// TwinCAT 3 PLC project Nepionic_Log
// Title: Nepionic_Log
// Company: Nepionic
// Author: Nepionic
// ProjectVersion: 0.1.1
// ProgramVersion: 3.1.4026.22
// libraries:
//   Tc2_Standard, * (Beckhoff Automation GmbH)
//   Tc2_System, * (Beckhoff Automation GmbH)
//   Tc2_Utilities, * (Beckhoff Automation GmbH)
//   Tc3_DynamicMemory, * (Beckhoff Automation GmbH)
// project tree:
//   Lib/Appenders/AdsLog/ AdsLogAppender.TcPOU (not stored), LogLevelToAdsLogMsgType.TcPOU
//   Lib/Appenders/File/ DeleteFilesState.TcDUT (not stored), DeleteOldFiles.TcPOU, GenerateTimeData.TcPOU (not stored), GetFileAgeInSeconds.TcPOU (not stored), LoggingConfiguration.TcDUT, PersistToFileState.TcDUT (not stored), RollingIntervals.TcDUT (not stored)
//   Lib/Appenders/ LogAppender.TcIO (not stored)
//   Lib/ Constants.TcGVL, DateTime.TcPOU (not stored), Error.TcDUT (not stored), ErrorCodes.TcDUT (not stored)
//   Lib/Core/ LogAttribute.TcDUT, LogAttributeType.TcDUT (not stored), LogAttributeValueToString.TcPOU, LogLevel.TcDUT
//   Lib/Manager/ GetLogManager.TcPOU (not stored), LogManager.TcPOU (not stored)
//   Lib/Logger/ DefaultLogger.TcPOU, Logger.TcIO (not stored)
//   Lib/String/ AnyToString.TcPOU (not stored), DefaultStringBuilder.TcPOU (not stored), DynamicStringBuffer.TcPOU (not stored), LimitedStringBuilder.TcIO (not stored), StringBuilder.TcIO (not stored)

// ---- Lib/Appenders/File/LoggingConfiguration.TcDUT
// Configuration of TcLogCore
TYPE LoggingConfiguration :
STRUCT
	// File name where the logs should be written to. Should not include path.
	file_name : Tc2_System.T_MaxString;
	// File path where the logs should be written to. Will be prefixed to `FileName`
	file_path : Tc2_System.T_MaxString;
	// Whether to include the instance path of TcLog into the log message or not.
	include_instance_path : BOOL;
	/// Whether to write the logs to ADS output or not.
	write_to_ads : BOOL;
	/// Rolling interval: when to create a new log file.
	rolling_interval : RollingIntervals;
	/// What is the minimum log level that gets logged?
	minimum_level : LogLevel;
	/// Which delimiter should be used between the different parts of the log string?
	delimiter : STRING(1);
	/// When should old log files be deleted? Unit: days. Set it to `0` if log files should never be deleted. 
	log_file_life_span : UINT;
	/// Format of timestamp. See `TcLogCore.TimestampFormat` for formatting options.
	timestamp_format : STRING;
	/// Log only valid timestamps (skip log messages during time initialization (first few cycles)
	valid_timestamps_only: BOOL;
END_STRUCT
END_TYPE

// ---- Lib/Core/LogAttribute.TcDUT
// A single structured log attribute attached to a log entry.
//
// Binary layout (96 bytes, little-endian, matched by the Go otelcol-ads parser):
//   offset  0..31   key         STRING(31)            = 32 bytes  attribute name
//   offset 32       attr_type   LogAttributeType      =  1 byte   type tag
//   offset 33..95   value_bytes ARRAY[0..62] BYTE     = 63 bytes  payload (see attr_type)
//
// For attr_type = LogAttributeType.Str (11):
//   value_bytes holds a null-terminated STRING(62).
// For numeric/bool types, value_bytes[0..N-1] holds the value as little-endian bytes.
TYPE LogAttribute :
STRUCT
	// Attribute name, e.g. 'event.name', 'axis.speed'
	key : STRING(31);
	
	// Type tag — one of the LogAttrType enum values.
	attr_type : LogAttributeType;

	// Raw value bytes. Interpretation depends on attr_type.
	// For String: null-terminated string up to 62 chars.
	// For numeric/bool: little-endian encoded value in first N bytes.
	value_bytes : ARRAY[0..62] OF BYTE;
END_STRUCT
END_TYPE

// ---- Lib/Core/LogLevel.TcDUT
{attribute 'qualified_only'}
{attribute 'strict'}
{attribute 'to_string'}
TYPE LogLevel :
(
	Debug := 0,
	Information := 1,
	Warning := 2,
	Error := 3,
	Fatal := 4
);
END_TYPE

// ---- Lib/Constants.TcGVL
{attribute 'qualified_only'}
VAR_GLOBAL CONSTANT
	/// Fifo overhead needed to manage the string buffer
	FifoOverhead : UDINT := 10;
	/// Buffer size of temporary buffer used to persist all log messages in one cycle. 
	BufferSize : UDINT := (100 * (Tc2_System.MAX_STRING_LENGTH + FifoOverhead));
END_VAR

// ---- Lib/Appenders/AdsLog/LogLevelToAdsLogMsgType.TcPOU
// Converts TcLog.LogLevels into Tc2_System.AdsLog_MsgType_*.
{attribute 'hide'}
FUNCTION INTERNAL LogLevelToAdsLogMsgType : DWORD
VAR_INPUT
	log_level : LogLevel;
END_VAR
VAR
	return_value : DWORD;
END_VAR

CASE log_level OF
	LogLevel.Debug, LogLevel.Information:
		return_value := Tc2_System.AdsLog_MsgType_Hint;
		
	LogLevel.Warning:
		return_value := Tc2_System.AdsLog_MsgType_Warn;
		
	LogLevel.Error, LogLevel.Fatal:
		return_value := Tc2_System.AdsLog_MsgType_Error;
ELSE
	return_value := Tc2_System.AdsLog_MsgType_Hint;
END_CASE

LogLevelToAdsLogMsgType := return_value;

END_FUNCTION

// ---- Lib/Appenders/File/DeleteOldFiles.TcPOU
{attribute 'hide_all_locals'}
FUNCTION_BLOCK INTERNAL DeleteOldFiles
VAR_INPUT
	StartScan : BOOL; // Rising edge starts scan for out-of-date log files and deletes them.
	ExpirationInDays : UINT; // Files will be deleted if older than n days
	FilePath : Tc2_System.T_MaxString; // Path to files to be deleted
	FileName : Tc2_System.T_MaxString; // Only files which match this filename will be deleted
	current_utc_time : Tc2_Utilities.T_FileTime; // Current time  as UTC
END_VAR
VAR_OUTPUT
	Error : Error; // Error information
END_VAR
VAR CONSTANT
	OneDayInSeconds : LREAL := 24*3600.0;
	MaxNumberOfFiles : UDINT := 100;
END_VAR
VAR
	_state : DeleteFilesState := DeleteFilesState.Idle;
	
	_enumFindFileList : Tc2_Utilities.Fb_EnumFindFileList;
	_enumBusy : Tc2_Standard.F_Trig;
	_fileDelete : Tc2_System.Fb_FileDelete;
	_fileDeleteBusy : Tc2_Standard.F_TRIG;
	_listOfFiles : ARRAY[1..100] OF Tc2_Utilities.St_FindFileEntry;
	_deleteFileIndex : UDINT;
	_fileNameToDelete : Tc2_System.T_MaxString;
	_commandType : Tc2_Utilities.E_EnumCmdType;
	_fileDeleted : BOOL;
	_startFileDelete: BOOL;
END_VAR

// State machine to delete all due files.
// It first enumerates all files in the specified directory
// and then deletes all files that have overpassed the specified due date
_startFileDelete := FALSE;

CASE _state OF
	DeleteFilesState.Idle:
		IF StartScan THEN
			_commandType := Tc2_Utilities.E_EnumCmdType.eEnumCmd_First;
			_deleteFileIndex := 1;
			_state := DeleteFilesState.SearchNextFile;
		END_IF
    
	DeleteFilesState.SearchNextFile:
		IF _enumBusy.Q THEN
			_state := DeleteFilesState.WaitUntilExecutionDone;
		END_IF
    
	DeleteFilesState.WaitUntilExecutionDone:
		IF NOT _enumFindFileList.bError THEN
			IF NOT _enumFindFileList.bEOE THEN
				IF _enumFindFileList.nFindFiles < MaxNumberOfFiles THEN
					_state := DeleteFilesState.SearchNextFile;
				ELSE
					_commandType := Tc2_Utilities.E_EnumCmdType.eEnumCmd_Abort;
				_state := DeleteFilesState.ProcessFoundFiles;
				END_IF
			ELSE
				_state := DeleteFilesState.ProcessFoundFiles;
			END_IF
		ELSE
		_state := DeleteFilesState.Idle;
		END_IF
    
	DeleteFilesState.ProcessFoundFiles:
		IF _deleteFileIndex > _enumFindFileList.nFindFiles THEN
			_state := DeleteFilesState.Idle;
		ELSE
			_state := DeleteFilesState.CheckIfFileIsDirectory;
		END_IF
    
	DeleteFilesState.CheckIfFileIsDirectory:
		IF NOT _listOfFiles[_deleteFileIndex].fileAttributes.bDirectory THEN
			_state := DeleteFilesState.CheckFileTime;
		ELSE
			_deleteFileIndex := _deleteFileIndex + 1;
			_state := DeleteFilesState.ProcessFoundFiles;
		END_IF
    
	DeleteFilesState.CheckFileTime:   
		IF GetFileAgeInSeconds(current_utc_time, _listOfFiles[_deleteFileIndex]) > (ExpirationInDays * OneDayInSeconds) THEN
			_state := DeleteFilesState.DeleteFile;
		ELSE
			_deleteFileIndex := _deleteFileIndex + 1;
			_state := DeleteFilesState.ProcessFoundFiles;
		END_IF
  
	DeleteFilesState.DeleteFile:
		_fileNameToDelete := Tc2_Standard.CONCAT(FilePath, _listOfFiles[_deleteFileIndex].sFileName);
		_startFileDelete := TRUE;
		
		IF _fileDeleteBusy.Q THEN
			_deleteFileIndex := _deleteFileIndex + 1;
			_fileDeleted := TRUE;
			_state := DeleteFilesState.FileDeleted;
		END_IF
		
		IF _fileDelete.bError THEN
			_state := DeleteFilesState.Idle;
		END_IF
    
	DeleteFilesState.FileDeleted:   
		// This state is needed to generate a rising edge for FB_FileDelete
		IF NOT _fileDeleted THEN
			_state := DeleteFilesState.ProcessFoundFiles;
		END_IF
		_fileDeleted := FALSE;
END_CASE

// Function blocks used in state machine

// Search files in given directory
_enumFindFileList(sNetId := '',
	eCmd := _commandType,
	sPathName := Tc2_Standard.CONCAT(FilePath, Tc2_Standard.CONCAT('*', FileName)),
	bExecute := (_state = DeleteFilesState.SearchNextFile)
		OR (
			_commandType = Tc2_Utilities.E_EnumCmdType.eEnumCmd_Abort
			AND _state <> DeleteFilesState.Idle
		),
	pFindList := ADR(_listOfFiles),
	cbFindList := SIZEOF(_listOfFiles),
	tTimeout := T#10S
);

_enumBusy(Clk := _enumFindFileList.bBusy);

// Delete files
_fileDelete(sNetId := '',
	sPathName := _fileNameToDelete,
	bExecute := _startFileDelete,
	tTimeout := T#10S
);

_fileDeleteBusy(Clk := _fileDelete.bBusy);

// Error handling
Error.Active := FALSE;
Error.Code := ErrorCodes.None;
Error.Info := '';

IF _enumFindFileList.bError THEN
	Error.Active := TRUE;
	Error.Code := ErrorCodes.EnumeratingFilesInSpecifiedDirectoryFailed;
	Error.Info := Tc2_Standard.Concat('Enumerating files in specified directory failed. Error thrown by FB_EnumFindFileList. Consult Beckhoff InfoSys. Internal Error: ', UDINT_TO_STRING(_enumFindFileList.nErrId));
END_IF

IF _fileDelete.bError THEN
	Error.Active := TRUE;
	Error.Code := ErrorCodes.DeletingFileFailed;
	Error.Info := Tc2_Standard.Concat('Deleting expired log file in specified directory failed. Error thrown by FB_FileDelete. Consult Beckhoff InfoSys. Internal Error: ', UDINT_TO_STRING(_fileDelete.nErrId));
END_IF

END_FUNCTION_BLOCK

// ---- Lib/Core/LogAttributeValueToString.TcPOU
/// Formats the value of a log attribute as a human-readable string.
///
/// Reads `value_bytes` according to `attr_type` and returns a string
/// representation suitable for embedding in log messages.
/// Numeric types are formatted with the standard TwinCAT `*_TO_STRING`
/// conversions; booleans become `'TRUE'` or `'FALSE'`; strings are
/// returned as-is (null terminator stripped by assignment).
FUNCTION PUBLIC LogAttributeValueToString : STRING(62)
VAR_IN_OUT
	attr : LogAttribute;
END_VAR
VAR
	base      : PVOID;
	sint_ptr  : POINTER TO SINT;
	int_ptr   : POINTER TO INT;
	dint_ptr  : POINTER TO DINT;
	lint_ptr  : POINTER TO LINT;
	usint_ptr : POINTER TO USINT;
	uint_ptr  : POINTER TO UINT;
	udint_ptr : POINTER TO UDINT;
	ulint_ptr : POINTER TO ULINT;
	real_ptr  : POINTER TO REAL;
	lreal_ptr : POINTER TO LREAL;
	str_ptr   : POINTER TO STRING(62);
END_VAR

// All typed pointers alias the same first byte of value_bytes — no copies needed.
base    := ADR(attr.value_bytes[0]);
sint_ptr  := base;
int_ptr   := base;
dint_ptr  := base;
lint_ptr  := base;
usint_ptr := base;
uint_ptr  := base;
udint_ptr := base;
ulint_ptr := base;
real_ptr  := base;
lreal_ptr := base;
str_ptr   := base;

CASE attr.attr_type OF
	LogAttributeType.Str:     LogAttributeValueToString := str_ptr^;
	LogAttributeType.Boolean: LogAttributeValueToString := SEL(attr.value_bytes[0] <> 0, 'FALSE', 'TRUE');
	LogAttributeType.Int8:    LogAttributeValueToString := SINT_TO_STRING(sint_ptr^);
	LogAttributeType.Int16:   LogAttributeValueToString := INT_TO_STRING(int_ptr^);
	LogAttributeType.Int32:   LogAttributeValueToString := DINT_TO_STRING(dint_ptr^);
	LogAttributeType.Int64:   LogAttributeValueToString := LINT_TO_STRING(lint_ptr^);
	LogAttributeType.UInt8:   LogAttributeValueToString := USINT_TO_STRING(usint_ptr^);
	LogAttributeType.UInt16:  LogAttributeValueToString := UINT_TO_STRING(uint_ptr^);
	LogAttributeType.UInt32:  LogAttributeValueToString := UDINT_TO_STRING(udint_ptr^);
	LogAttributeType.UInt64:  LogAttributeValueToString := ULINT_TO_STRING(ulint_ptr^);
	LogAttributeType.Float32: LogAttributeValueToString := REAL_TO_STRING(real_ptr^);
	LogAttributeType.Float64: LogAttributeValueToString := LREAL_TO_STRING(lreal_ptr^);
ELSE
	LogAttributeValueToString := '(unknown)';
END_CASE

END_FUNCTION

// ---- Lib/Logger/DefaultLogger.TcPOU
/// Concrete logger that dispatches to the process-global `LogManager` singleton.
///
/// Declare one instance per component/axis/subsystem and pass `name` to
/// `FB_Init` — the name becomes the `source` field on every log record so
/// you can filter by component in your log viewer.
///
/// Simple usage:
/// ```st
/// VAR
///   log : DefaultLogger('AxisX');
/// END_VAR
/// log.Info('Homing started');
/// log.Error('Limit switch triggered');
/// ```
///
/// Structured attributes and conditional logging:
/// ```st
/// log.WithAttribute('state', 'Homing').WithAttribute('speed', '100').Info('Axis moving');
/// log.OnCondition(error_active).Error('Drive fault detected');
/// ```
///
/// No wiring required — `FB_Init` connects automatically to `GetLogManager()`.
/// Register appenders on `GetLogManager()` once at program startup.
{attribute 'linkalways'}
{attribute 'no_explicit_call' := 'This FB is a CLASS and must be accessed using methods or properties'}
{attribute 'enable_dynamic_creation'}
{attribute 'reflection'}
FUNCTION_BLOCK PUBLIC DefaultLogger IMPLEMENTS Logger
VAR
	{attribute 'instance-path'}
    {attribute 'noinit'}
    instance_path : STRING(255);
	
	_name : STRING(255);
	attributes : ARRAY[0..9] OF LogAttribute;
	attribute_count : USINT;
	condition : BOOL := TRUE;
	chain_started : BOOL;
END_VAR
VAR CONSTANT
	INSTANCE_PATH_KEY_NAME : STRING := 'instance_path';
END_VAR

/// Log at DEBUG level.
METHOD PUBLIC Debug : BOOL
VAR_INPUT
	message : Tc2_System.T_MaxString;
END_VAR
InitChain();
IF condition THEN
	GetLogManager().Dispatch(LogLevel.Debug, message, _name, attributes, attribute_count);
END_IF
ResetChain();
Debug := TRUE;
END_METHOD

/// Log at ERROR level.
METHOD PUBLIC Error : BOOL
VAR_INPUT
	message : Tc2_System.T_MaxString;
END_VAR
InitChain();
IF condition THEN
	GetLogManager().Dispatch(LogLevel.Error, message, _name, attributes, attribute_count);
END_IF
ResetChain();
Error := TRUE;
END_METHOD

/// Log at FATAL level.
METHOD PUBLIC Fatal : BOOL
VAR_INPUT
	message : Tc2_System.T_MaxString;
END_VAR
InitChain();
IF condition THEN
	GetLogManager().Dispatch(LogLevel.Fatal, message, _name, attributes, attribute_count);
END_IF
ResetChain();
Fatal := TRUE;
END_METHOD

METHOD FB_Init : BOOL
VAR_INPUT
	bInitRetains : BOOL;
	bInCopyCode : BOOL;
	/// Component name used as the `source` field on every log record.
	name : STRING(63);
END_VAR
_name := name;
END_METHOD

/// Log at INFORMATION level.
METHOD PUBLIC Info : BOOL
VAR_INPUT
	message : Tc2_System.T_MaxString;
END_VAR
InitChain();
IF condition THEN
	GetLogManager().Dispatch(LogLevel.Information, message, _name, attributes, attribute_count);
END_IF
ResetChain();
Info := TRUE;
END_METHOD

// Initialise chain state on the first call of a log chain.
// Idempotent — safe to call from every chain method.
{attribute 'hide'}
METHOD PRIVATE InitChain
IF NOT chain_started THEN
	chain_started := TRUE;
	condition := TRUE;
	attribute_count := 0;
END_IF
END_METHOD

/// Component name used as the `source` field on every log record.
{attribute 'monitoring' := 'call'}
PROPERTY PUBLIC Name : STRING(63)
GET // PUBLIC
Name := _name;
END_GET
SET // PUBLIC
_name := Name;
END_SET
END_PROPERTY

/// Conditionally emit the log record.
/// When `cond` is FALSE the chain is still initialised but the terminal
/// method (`Debug`, `Info`, etc.) will be a no-op.
/// ```st
/// log.OnCondition(error_active).Error('Drive fault');
/// ```
METHOD PUBLIC OnCondition : REFERENCE TO DefaultLogger
VAR_INPUT
	cond : BOOL;
END_VAR
InitChain();
condition := cond;
OnCondition REF= THIS^;
END_METHOD

// Reset chain state after a terminal method completes.
// Must be called at the end of every Debug/Info/Warning/Error/Fatal implementation.
{attribute 'hide'}
METHOD PRIVATE ResetChain
chain_started := FALSE;
condition := TRUE;
attribute_count := 0;
END_METHOD

/// Log at WARNING level.
METHOD PUBLIC Warning : BOOL
VAR_INPUT
	message : Tc2_System.T_MaxString;
END_VAR
InitChain();
IF condition THEN
	GetLogManager().Dispatch(LogLevel.Warning, message, _name, attributes, attribute_count);
END_IF
ResetChain();
Warning := TRUE;
END_METHOD

/// Attach a string key/value attribute to the current log record.
/// Call before the terminal method (`Debug`, `Info`, `Warning`, `Error`, `Fatal`).
/// Up to 10 attributes per record; extras are silently ignored.
/// Chainable:
/// ```st
/// log.WithAttribute('state', 'Homing').WithDIntAttribute('pos', position).Info('Moving');
/// ```
METHOD PUBLIC WithAttribute : REFERENCE TO DefaultLogger
VAR_INPUT
	key : STRING(31);
	value : STRING(62);
END_VAR
InitChain();

IF attribute_count < 10 THEN
	attributes[attribute_count].key := key;
	attributes[attribute_count].attr_type := LogAttributeType.Str;
	Tc2_System.MemCpy(ADR(attributes[attribute_count].value_bytes[0]), ADR(value), SIZEOF(STRING(62)));
	attribute_count := attribute_count + 1;
END_IF

WithAttribute REF= THIS^;
END_METHOD

/// Attach a BOOL attribute.
METHOD PUBLIC WithBoolAttribute : REFERENCE TO DefaultLogger
VAR_INPUT
	key : STRING(31);
	value : BOOL;
END_VAR
InitChain();

IF attribute_count < 10 THEN
	attributes[attribute_count].key := key;
	attributes[attribute_count].attr_type := LogAttributeType.Boolean;
	attributes[attribute_count].value_bytes[0] := BOOL_TO_BYTE(value);
	attribute_count := attribute_count + 1;
END_IF

WithBoolAttribute REF= THIS^;
END_METHOD

/// Attach a DINT (32-bit signed) attribute.
METHOD PUBLIC WithDIntAttribute : REFERENCE TO DefaultLogger
VAR_INPUT
	key : STRING(31);
	value : DINT;
END_VAR
InitChain();

IF attribute_count < 10 THEN
	attributes[attribute_count].key := key;
	attributes[attribute_count].attr_type := LogAttributeType.Int32;
	Tc2_System.MemCpy(ADR(attributes[attribute_count].value_bytes[0]), ADR(value), SIZEOF(DINT));
	attribute_count := attribute_count + 1;
END_IF

WithDIntAttribute REF= THIS^;
END_METHOD

/// Attach the instance path to the current log record.
/// Call before the terminal method (`Debug`, `Info`, `Warning`, `Error`, `Fatal`).
/// Chainable:
/// ```st
/// log.WithInstancePath().WithDIntAttribute('pos', position).Info('Moving');
/// ```
METHOD PUBLIC WithInstancePath : REFERENCE TO DefaultLogger
WithInstancePath REF= WithAttribute(INSTANCE_PATH_KEY_NAME, instance_path);
END_METHOD

/// Attach an INT (16-bit signed) attribute.
METHOD PUBLIC WithIntAttribute : REFERENCE TO DefaultLogger
VAR_INPUT
	key : STRING(31);
	value : INT;
END_VAR
InitChain();

IF attribute_count < 10 THEN
	attributes[attribute_count].key := key;
	attributes[attribute_count].attr_type := LogAttributeType.Int16;
	Tc2_System.MemCpy(ADR(attributes[attribute_count].value_bytes[0]), ADR(value), SIZEOF(INT));
	attribute_count := attribute_count + 1;
END_IF

WithIntAttribute REF= THIS^;
END_METHOD

/// Attach a LINT (64-bit signed) attribute.
METHOD PUBLIC WithLIntAttribute : REFERENCE TO DefaultLogger
VAR_INPUT
	key : STRING(31);
	value : LINT;
END_VAR
InitChain();

IF attribute_count < 10 THEN
	attributes[attribute_count].key := key;
	attributes[attribute_count].attr_type := LogAttributeType.Int64;
	Tc2_System.MemCpy(ADR(attributes[attribute_count].value_bytes[0]), ADR(value), SIZEOF(LINT));
	attribute_count := attribute_count + 1;
END_IF

WithLIntAttribute REF= THIS^;
END_METHOD

/// Attach an LREAL (64-bit float) attribute.
METHOD PUBLIC WithLRealAttribute : REFERENCE TO DefaultLogger
VAR_INPUT
	key : STRING(31);
	value : LREAL;
END_VAR
InitChain();

IF attribute_count < 10 THEN
	attributes[attribute_count].key := key;
	attributes[attribute_count].attr_type := LogAttributeType.Float64;
	Tc2_System.MemCpy(ADR(attributes[attribute_count].value_bytes[0]), ADR(value), SIZEOF(LREAL));
	attribute_count := attribute_count + 1;
END_IF

WithLRealAttribute REF= THIS^;
END_METHOD

/// Attach a REAL (32-bit float) attribute.
METHOD PUBLIC WithRealAttribute : REFERENCE TO DefaultLogger
VAR_INPUT
	key : STRING(31);
	value : REAL;
END_VAR
InitChain();

IF attribute_count < 10 THEN
	attributes[attribute_count].key := key;
	attributes[attribute_count].attr_type := LogAttributeType.Float32;
	Tc2_System.MemCpy(ADR(attributes[attribute_count].value_bytes[0]), ADR(value), SIZEOF(REAL));
	attribute_count := attribute_count + 1;
END_IF

WithRealAttribute REF= THIS^;
END_METHOD

/// Attach a UDINT (32-bit unsigned) attribute.
METHOD PUBLIC WithUDIntAttribute : REFERENCE TO DefaultLogger
VAR_INPUT
	key : STRING(31);
	value : UDINT;
END_VAR
InitChain();

IF attribute_count < 10 THEN
	attributes[attribute_count].key := key;
	attributes[attribute_count].attr_type := LogAttributeType.Uint32;
	Tc2_System.MemCpy(ADR(attributes[attribute_count].value_bytes[0]), ADR(value), SIZEOF(UDINT));
	attribute_count := attribute_count + 1;
END_IF

WithUDIntAttribute REF= THIS^;
END_METHOD

/// Attach a UINT (16-bit unsigned) attribute.
METHOD PUBLIC WithUIntAttribute : REFERENCE TO DefaultLogger
VAR_INPUT
	key : STRING(31);
	value : UINT;
END_VAR
InitChain();

IF attribute_count < 10 THEN
	attributes[attribute_count].key := key;
	attributes[attribute_count].attr_type := LogAttributeType.Uint16;
	Tc2_System.MemCpy(ADR(attributes[attribute_count].value_bytes[0]), ADR(value), SIZEOF(UINT));
	attribute_count := attribute_count + 1;
END_IF

WithUIntAttribute REF= THIS^;
END_METHOD

/// Attach a ULINT (64-bit unsigned) attribute.
METHOD PUBLIC WithULIntAttribute : REFERENCE TO DefaultLogger
VAR_INPUT
	key : STRING(31);
	value : ULINT;
END_VAR
InitChain();

IF attribute_count < 10 THEN
	attributes[attribute_count].key := key;
	attributes[attribute_count].attr_type := LogAttributeType.Uint64;
	Tc2_System.MemCpy(ADR(attributes[attribute_count].value_bytes[0]), ADR(value), SIZEOF(ULINT));
	attribute_count := attribute_count + 1;
END_IF

WithULIntAttribute REF= THIS^;
END_METHOD

END_FUNCTION_BLOCK
